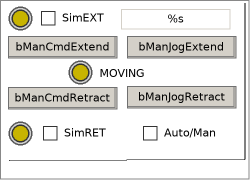
VISUALIZATION Piston  // 250x180
VAR_IN_OUT
	piston : ST_HmiPiston;
END_VAR
    Lamp1 (6,5 29x27), variable: piston.bIsExtended, style: Lamp-Lamp1-Yellow
    Button (8,36 109x22), "bManCmdExtend"
        tap piston.bManCmdExtend
    Button (127,36 109x22), "bManJogExtend"
        tap piston.bManJogExtend
    Button (127,86 109x22), "bManJogRetract"
        tap piston.bManJogRetract
    Button (8,87 109x22), "bManCmdRetract"
        tap piston.bManCmdRetract
    Textfield (121,9 109x20), "%s", text variable: piston.Name
    Lamp1 (6,120 29x27), variable: piston.bIsRetracted, style: Lamp-Lamp1-Yellow
    Label (69,62 106x23), "MOVING", invisible if: NOT(piston.bIsMoving)
    Lamp1 (66,59 29x27), variable: piston.bOutSolenoidExtend, style: Lamp-Lamp1-Yellow
    Checkbox (141,118 100x30), "Auto/Man", variable: piston.bMode
    Checkbox (41,118 84x30), "SimRET", variable: piston.bSimulateRetracted
    Checkbox (39,3 84x30), "SimEXT", variable: piston.bSimulateExtended
    Line (9,160) (244,159)
    Line (245,159) (245,3)
END_VISUALIZATION

(* stored: Version 1.1.0.1, ProductVersion 3.1.4024.16
   Visu Piston: Id {9fd7dbe0-434c-4eae-a1d5-37e7a78ef247} *)
